ABB RAPID module: 001956CB

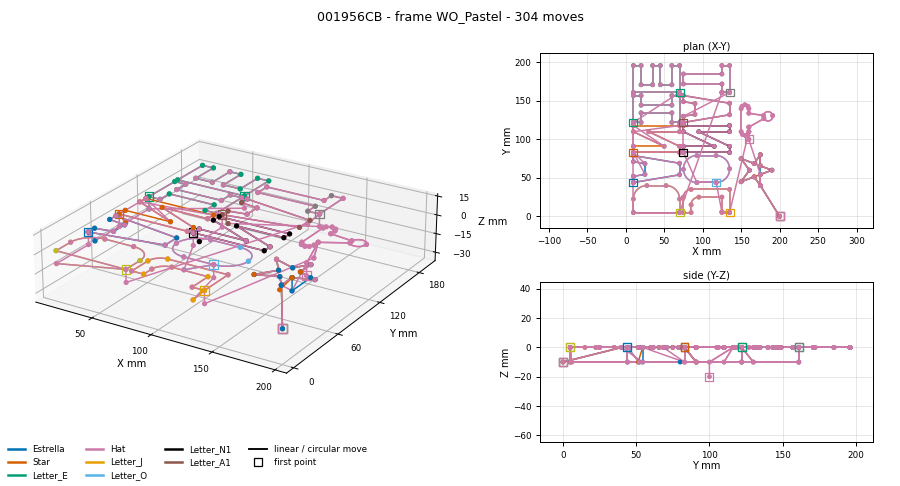
[picture p0: tool path of 001956CB in frame WO_Pastel, 304 of 314 moves have a stored position in this frame; points joined in program order, loops and branches not executed]
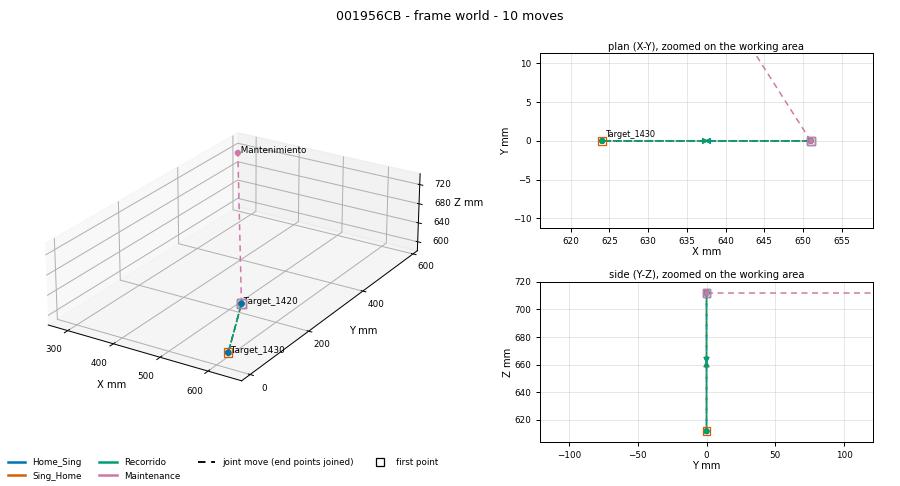
[picture p1: tool path of 001956CB in frame world, 10 of 314 moves have a stored position in this frame; points joined in program order, loops and branches not executed]
MODULE Module1
        CONST robtarget Target_10:=[[200,0,-10],[1,0,0,0],[0,0,2,0],[9E+09,9E+09,9E+09,9E+09,9E+09,9E+09]];
    CONST robtarget Target_20:=[[175,40,0],[1,0,0,0],[0,0,2,0],[9E+09,9E+09,9E+09,9E+09,9E+09,9E+09]];
    CONST robtarget Target_30:=[[175,54.375,0],[1,0,0,0],[0,0,2,0],[9E+09,9E+09,9E+09,9E+09,9E+09,9E+09]];
    CONST robtarget Target_40:=[[190,60,0],[1,0,0,0],[0,0,2,0],[9E+09,9E+09,9E+09,9E+09,9E+09,9E+09]];
    CONST robtarget Target_50:=[[175,65.625,0],[1,0,0,0],[0,0,2,0],[9E+09,9E+09,9E+09,9E+09,9E+09,9E+09]];
    CONST robtarget Target_60:=[[175,80,0],[1,0,0,0],[0,0,2,0],[9E+09,9E+09,9E+09,9E+09,9E+09,9E+09]];
    CONST robtarget Target_70:=[[166.901,68.662,0],[1,0,0,0],[0,0,2,0],[9E+09,9E+09,9E+09,9E+09,9E+09,9E+09]];
    CONST robtarget Target_80:=[[150,75,0],[1,0,0,0],[0,0,2,0],[9E+09,9E+09,9E+09,9E+09,9E+09,9E+09]];
    CONST robtarget Target_90:=[[160.714,60,0],[1,0,0,0],[0,0,2,0],[9E+09,9E+09,9E+09,9E+09,9E+09,9E+09]];
    CONST robtarget Target_100:=[[150,45,0],[1,0,0,0],[0,0,2,0],[9E+09,9E+09,9E+09,9E+09,9E+09,9E+09]];
    CONST robtarget Target_110:=[[166.901,51.338,0],[1,0,0,0],[0,0,2,0],[9E+09,9E+09,9E+09,9E+09,9E+09,9E+09]];
    CONST robtarget Target_120:=[[166.901,51.338,-10],[1,0,0,0],[-1,-1,2,0],[9E+09,9E+09,9E+09,9E+09,9E+09,9E+09]];
    CONST robtarget Target_130:=[[160,116,0],[1,0,0,0],[0,0,2,0],[9E+09,9E+09,9E+09,9E+09,9E+09,9E+09]];
    CONST robtarget Target_140:=[[179.71,127.038,0],[1,0,0,0],[0,0,2,0],[9E+09,9E+09,9E+09,9E+09,9E+09,9E+09]];
    CONST robtarget Target_150:=[[186.774,124.203,0],[1,0,0,0],[0,0,2,0],[9E+09,9E+09,9E+09,9E+09,9E+09,9E+09]];
    CONST robtarget Target_160:=[[190.983,130.98,0],[1,0,0,0],[0,0,2,0],[9E+09,9E+09,9E+09,9E+09,9E+09,9E+09]];
    CONST robtarget Target_170:=[[183.755,135.933,0],[1,0,0,0],[0,0,2,0],[9E+09,9E+09,9E+09,9E+09,9E+09,9E+09]];
    CONST robtarget Target_180:=[[179.014,130.957,0],[1,0,0,0],[0,0,2,0],[9E+09,9E+09,9E+09,9E+09,9E+09,9E+09]];
    CONST robtarget Target_190:=[[160,134,0],[1,0,0,0],[0,0,2,0],[9E+09,9E+09,9E+09,9E+09,9E+09,9E+09]];
    CONST robtarget Target_200:=[[160,140,0],[1,0,0,0],[0,0,2,0],[9E+09,9E+09,9E+09,9E+09,9E+09,9E+09]];
    CONST robtarget Target_210:=[[158.829,143.215,0],[1,0,0,0],[0,0,2,0],[9E+09,9E+09,9E+09,9E+09,9E+09,9E+09]];
    CONST robtarget Target_220:=[[154.832,144.997,0],[1,0,0,0],[0,0,2,0],[9E+09,9E+09,9E+09,9E+09,9E+09,9E+09]];
    CONST robtarget Target_230:=[[151.042,143.055,0],[1,0,0,0],[0,0,2,0],[9E+09,9E+09,9E+09,9E+09,9E+09,9E+09]];
        CONST robtarget HomeManipulador:=[[651,-0.02,712.04],[0.707129,-3.57758E-05,0.707084,6.57305E-06],[0,0,-1,0],[9E+09,9E+09,9E+09,9E+09,9E+09,9E+09]];
    CONST robtarget Target_1280:=[[70,161,0],[1,0,0,0],[-1,-2,-1,0],[9E+09,9E+09,9E+09,9E+09,9E+09,9E+09]];
    CONST robtarget Target_1290:=[[70,196,0],[1,0,0,0],[-1,-2,-1,0],[9E+09,9E+09,9E+09,9E+09,9E+09,9E+09]];
    CONST robtarget Target_1300:=[[60,196,0],[1,0,0,0],[-1,-2,-1,0],[9E+09,9E+09,9E+09,9E+09,9E+09,9E+09]];
    CONST robtarget Target_1310:=[[60,171,0],[1,0,0,0],[-1,-2,-1,0],[9E+09,9E+09,9E+09,9E+09,9E+09,9E+09]];
    CONST robtarget Target_1320:=[[45,171,0],[1,0,0,0],[-1,-2,-1,0],[9E+09,9E+09,9E+09,9E+09,9E+09,9E+09]];
    CONST robtarget Target_1330:=[[45,196,0],[1,0,0,0],[-1,-2,-1,0],[9E+09,9E+09,9E+09,9E+09,9E+09,9E+09]];
    CONST robtarget Target_1340:=[[35,196,0],[1,0,0,0],[-1,-2,-1,0],[9E+09,9E+09,9E+09,9E+09,9E+09,9E+09]];
    CONST robtarget Target_1350:=[[35,171,0],[1,0,0,0],[-1,-2,-1,0],[9E+09,9E+09,9E+09,9E+09,9E+09,9E+09]];
    CONST robtarget Target_1360:=[[20,171,0],[1,0,0,0],[-1,-2,-1,0],[9E+09,9E+09,9E+09,9E+09,9E+09,9E+09]];
    CONST robtarget Target_1370:=[[20,196,0],[1,0,0,0],[-1,-2,-1,0],[9E+09,9E+09,9E+09,9E+09,9E+09,9E+09]];
    CONST robtarget Target_1380:=[[10,196,0],[1,0,0,0],[-1,-2,-1,0],[9E+09,9E+09,9E+09,9E+09,9E+09,9E+09]];
    CONST robtarget Target_1390:=[[10,161,0],[1,0,0,0],[-1,-2,-1,0],[9E+09,9E+09,9E+09,9E+09,9E+09,9E+09]];
    CONST robtarget Target_1470:=[[160,100.007,-20],[1,0,0,0],[0,2,0,1],[9E+09,9E+09,9E+09,9E+09,9E+09,9E+09]];
    CONST robtarget Target_1440:=[[160,100,-10],[1,0,0,0],[0,0,2,0],[9E+09,9E+09,9E+09,9E+09,9E+09,9E+09]];
    CONST robtarget Target_240:=[[150,140,0],[1,0,0,0],[0,0,2,0],[9E+09,9E+09,9E+09,9E+09,9E+09,9E+09]];
    CONST robtarget Target_250:=[[150,110,0],[1,0,0,0],[0,0,2,0],[9E+09,9E+09,9E+09,9E+09,9E+09,9E+09]];
    CONST robtarget Target_260:=[[151.712,106.233,0],[1,0,0,0],[0,-1,2,0],[9E+09,9E+09,9E+09,9E+09,9E+09,9E+09]];
    CONST robtarget Target_270:=[[155.472,105.022,0],[1,0,0,0],[0,0,2,0],[9E+09,9E+09,9E+09,9E+09,9E+09,9E+09]];
    CONST robtarget Target_280:=[[158.325,106.266,0],[1,0,0,0],[0,0,2,0],[9E+09,9E+09,9E+09,9E+09,9E+09,9E+09]];
    CONST robtarget Target_290:=[[160,110.007,0],[1,0,0,0],[0,0,2,0],[9E+09,9E+09,9E+09,9E+09,9E+09,9E+09]];
    CONST robtarget Target_300:=[[160,110.007,-10],[1,0,0,0],[0,0,2,0],[9E+09,9E+09,9E+09,9E+09,9E+09,9E+09]];
    CONST robtarget Target_310_2:=[[135,5,0],[1,0,0,0],[0,0,2,0],[9E+09,9E+09,9E+09,9E+09,9E+09,9E+09]];
    CONST robtarget Target_320_2:=[[135,35,0],[1,0,0,0],[0,0,2,0],[9E+09,9E+09,9E+09,9E+09,9E+09,9E+09]];
    CONST robtarget Target_330_2:=[[85,35,0],[1,0,0,0],[0,0,2,0],[9E+09,9E+09,9E+09,9E+09,9E+09,9E+09]];
    CONST robtarget Target_340_2:=[[77.06,31.078,0],[1,0,0,0],[0,0,2,0],[9E+09,9E+09,9E+09,9E+09,9E+09,9E+09]];
    CONST robtarget Target_350_2:=[[75,25,0],[1,0,0,0],[0,0,2,0],[9E+09,9E+09,9E+09,9E+09,9E+09,9E+09]];
    CONST robtarget Target_360_2:=[[75,5,0],[1,0,0,0],[0,0,2,0],[9E+09,9E+09,9E+09,9E+09,9E+09,9E+09]];
    CONST robtarget Target_370_2:=[[85,5,0],[1,0,0,0],[0,0,2,0],[9E+09,9E+09,9E+09,9E+09,9E+09,9E+09]];
    CONST robtarget Target_380_2:=[[85,15,0],[1,0,0,0],[0,0,2,0],[9E+09,9E+09,9E+09,9E+09,9E+09,9E+09]];
    CONST robtarget Target_390_2:=[[87.41,21.51,0],[1,0,0,0],[0,0,2,0],[9E+09,9E+09,9E+09,9E+09,9E+09,9E+09]];
    CONST robtarget Target_400_2:=[[95,25,0],[1,0,0,0],[0,0,2,0],[9E+09,9E+09,9E+09,9E+09,9E+09,9E+09]];
    CONST robtarget Target_410_2:=[[125,25,0],[1,0,0,0],[0,0,2,0],[9E+09,9E+09,9E+09,9E+09,9E+09,9E+09]];
    CONST robtarget Target_420_2:=[[125,5,0],[1,0,0,0],[0,0,2,0],[9E+09,9E+09,9E+09,9E+09,9E+09,9E+09]];
    CONST robtarget Target_430_2:=[[125,6,-10],[1,0,0,0],[0,0,2,0],[9E+09,9E+09,9E+09,9E+09,9E+09,9E+09]];
    CONST robtarget Target_440:=[[117.496,44,0],[1,0,0,0],[0,0,2,0],[9E+09,9E+09,9E+09,9E+09,9E+09,9E+09]];
    CONST robtarget Target_450:=[[130.812,50.14,0],[1,0,0,0],[0,0,2,0],[9E+09,9E+09,9E+09,9E+09,9E+09,9E+09]];
    CONST robtarget Target_460:=[[134.997,61.803,0],[1,0,0,0],[0,0,2,0],[9E+09,9E+09,9E+09,9E+09,9E+09,9E+09]];
    CONST robtarget Target_470:=[[131.095,72.519,0],[1,0,0,0],[0,0,2,0],[9E+09,9E+09,9E+09,9E+09,9E+09,9E+09]];
    CONST robtarget Target_490:=[[117.5,79,0],[1,0,0,0],[0,0,2,0],[9E+09,9E+09,9E+09,9E+09,9E+09,9E+09]];
    CONST robtarget Target_500:=[[92.5,79,0],[1,0,0,0],[0,0,2,0],[9E+09,9E+09,9E+09,9E+09,9E+09,9E+09]];
    CONST robtarget Target_510:=[[80.951,74.647,0],[1,0,0,0],[0,0,2,0],[9E+09,9E+09,9E+09,9E+09,9E+09,9E+09]];
    CONST robtarget Target_520:=[[75.005,61.068,0],[1,0,0,0],[0,0,2,0],[9E+09,9E+09,9E+09,9E+09,9E+09,9E+09]];
    CONST robtarget Target_530:=[[79.917,49.337,0],[1,0,0,0],[0,0,2,0],[9E+09,9E+09,9E+09,9E+09,9E+09,9E+09]];
    CONST robtarget Target_550:=[[92.504,44,0],[1,0,0,0],[0,0,2,0],[9E+09,9E+09,9E+09,9E+09,9E+09,9E+09]];
    CONST robtarget Target_560:=[[92.504,44,-10],[1,0,0,0],[0,0,2,0],[9E+09,9E+09,9E+09,9E+09,9E+09,9E+09]];
    CONST robtarget Target_570:=[[75,83,0],[1,0,0,0],[0,0,2,0],[9E+09,9E+09,9E+09,9E+09,9E+09,9E+09]];
    CONST robtarget Target_580:=[[135,83,0],[1,0,0,0],[0,0,2,0],[9E+09,9E+09,9E+09,9E+09,9E+09,9E+09]];
    CONST robtarget Target_590:=[[135,91,0],[1,0,0,0],[0,0,2,0],[9E+09,9E+09,9E+09,9E+09,9E+09,9E+09]];
    CONST robtarget Target_600:=[[95,110,0],[1,0,0,0],[0,0,2,0],[9E+09,9E+09,9E+09,9E+09,9E+09,9E+09]];
    CONST robtarget Target_610:=[[135,110,0],[1,0,0,0],[0,0,2,0],[9E+09,9E+09,9E+09,9E+09,9E+09,9E+09]];
    CONST robtarget Target_620:=[[135,118,0],[1,0,0,0],[0,0,2,0],[9E+09,9E+09,9E+09,9E+09,9E+09,9E+09]];
    CONST robtarget Target_630:=[[75,118,0],[1,0,0,0],[0,0,2,0],[9E+09,9E+09,9E+09,9E+09,9E+09,9E+09]];
    CONST robtarget Target_640:=[[75,110,0],[1,0,0,0],[0,0,2,0],[9E+09,9E+09,9E+09,9E+09,9E+09,9E+09]];
    CONST robtarget Target_650:=[[115,91,0],[1,0,0,0],[0,0,2,0],[9E+09,9E+09,9E+09,9E+09,9E+09,9E+09]];
    CONST robtarget Target_660:=[[75,91,0],[1,0,0,0],[0,0,2,0],[9E+09,9E+09,9E+09,9E+09,9E+09,9E+09]];
    CONST robtarget Target_670:=[[75,91,-10],[1,0,0,0],[0,0,2,0],[9E+09,9E+09,9E+09,9E+09,9E+09,9E+09]];
    CONST robtarget Target_680:=[[75,122,0],[1,0,0,0],[0,0,2,0],[9E+09,9E+09,9E+09,9E+09,9E+09,9E+09]];
    CONST robtarget Target_690:=[[135,132,0],[1,0,0,0],[0,0,2,0],[9E+09,9E+09,9E+09,9E+09,9E+09,9E+09]];
    CONST robtarget Target_700:=[[135,147,0],[1,0,0,0],[0,0,2,0],[9E+09,9E+09,9E+09,9E+09,9E+09,9E+09]];
    CONST robtarget Target_710:=[[75,157,0],[1,0,0,0],[0,0,2,0],[9E+09,9E+09,9E+09,9E+09,9E+09,9E+09]];
    CONST robtarget Target_720:=[[75,149,0],[1,0,0,0],[0,0,2,0],[9E+09,9E+09,9E+09,9E+09,9E+09,9E+09]];
    CONST robtarget Target_730:=[[90,146.5,0],[1,0,0,0],[0,0,2,0],[9E+09,9E+09,9E+09,9E+09,9E+09,9E+09]];
    CONST robtarget Target_740:=[[90,132.5,0],[1,0,0,0],[0,0,2,0],[9E+09,9E+09,9E+09,9E+09,9E+09,9E+09]];
    CONST robtarget Target_750:=[[75,130,0],[1,0,0,0],[0,0,2,0],[9E+09,9E+09,9E+09,9E+09,9E+09,9E+09]];
    CONST robtarget Target_760:=[[75,130,-10],[1,0,0,0],[0,0,2,0],[9E+09,9E+09,9E+09,9E+09,9E+09,9E+09]];
    CONST robtarget Target_770:=[[135,161,0],[1,0,0,0],[0,0,2,0],[9E+09,9E+09,9E+09,9E+09,9E+09,9E+09]];
    CONST robtarget Target_780:=[[135,196,0],[1,0,0,0],[0,0,2,0],[9E+09,9E+09,9E+09,9E+09,9E+09,9E+09]];
    CONST robtarget Target_790:=[[125,196,0],[1,0,0,0],[0,0,2,0],[9E+09,9E+09,9E+09,9E+09,9E+09,9E+09]];
    CONST robtarget Target_800:=[[125,185,0],[1,0,0,0],[0,0,2,0],[9E+09,9E+09,9E+09,9E+09,9E+09,9E+09]];
    CONST robtarget Target_810:=[[75,185,0],[1,0,0,0],[0,0,2,0],[9E+09,9E+09,9E+09,9E+09,9E+09,9E+09]];
    CONST robtarget Target_820:=[[75,172,0],[1,0,0,0],[0,0,2,0],[9E+09,9E+09,9E+09,9E+09,9E+09,9E+09]];
    CONST robtarget Target_830:=[[125,172,0],[1,0,0,0],[0,0,2,0],[9E+09,9E+09,9E+09,9E+09,9E+09,9E+09]];
    CONST robtarget Target_840:=[[125,161,0],[1,0,0,0],[0,0,2,0],[9E+09,9E+09,9E+09,9E+09,9E+09,9E+09]];
    CONST robtarget Target_850:=[[125,161,-10],[1,0,0,0],[0,0,2,0],[9E+09,9E+09,9E+09,9E+09,9E+09,9E+09]];
    CONST robtarget Target_860:=[[70,5,0],[1,0,0,0],[0,0,2,0],[9E+09,9E+09,9E+09,9E+09,9E+09,9E+09]];
    CONST robtarget Target_870:=[[70,22.489,0],[1,0,0,0],[0,0,2,0],[9E+09,9E+09,9E+09,9E+09,9E+09,9E+09]];
    CONST robtarget Target_880:=[[65.387,34.34,0],[1,0,0,0],[0,0,2,0],[9E+09,9E+09,9E+09,9E+09,9E+09,9E+09]];
    CONST robtarget Target_890:=[[52.5,40,0],[1,0,0,0],[0,0,2,0],[9E+09,9E+09,9E+09,9E+09,9E+09,9E+09]];
    CONST robtarget Target_900:=[[27.5,40,0],[1,0,0,0],[0,0,2,0],[9E+09,9E+09,9E+09,9E+09,9E+09,9E+09]];
    CONST robtarget Target_910:=[[14.273,33.958,0],[1,0,0,0],[0,0,2,0],[9E+09,9E+09,9E+09,9E+09,9E+09,9E+09]];
    CONST robtarget Target_920:=[[10,22.489,0],[1,0,0,0],[0,-1,2,0],[9E+09,9E+09,9E+09,9E+09,9E+09,9E+09]];
    CONST robtarget Target_930:=[[10,5,0],[1,0,0,0],[0,0,2,0],[9E+09,9E+09,9E+09,9E+09,9E+09,9E+09]];
    CONST robtarget Target_940:=[[10,5,-10],[1,0,0,0],[0,0,2,0],[9E+09,9E+09,9E+09,9E+09,9E+09,9E+09]];
    CONST robtarget Target_950:=[[10,44,0],[1,0,0,0],[0,0,2,0],[9E+09,9E+09,9E+09,9E+09,9E+09,9E+09]];
    CONST robtarget Target_960:=[[70,54,0],[1,0,0,0],[0,0,2,0],[9E+09,9E+09,9E+09,9E+09,9E+09,9E+09]];
    CONST robtarget Target_970:=[[70,69,0],[1,0,0,0],[0,0,2,0],[9E+09,9E+09,9E+09,9E+09,9E+09,9E+09]];
    CONST robtarget Target_980:=[[10,79,0],[1,0,0,0],[0,0,2,0],[9E+09,9E+09,9E+09,9E+09,9E+09,9E+09]];
    CONST robtarget Target_990:=[[10,71,0],[1,0,0,0],[0,0,2,0],[9E+09,9E+09,9E+09,9E+09,9E+09,9E+09]];
    CONST robtarget Target_1000:=[[25,68.5,0],[1,0,0,0],[0,0,2,0],[9E+09,9E+09,9E+09,9E+09,9E+09,9E+09]];
    CONST robtarget Target_1010:=[[25,54.5,0],[1,0,0,0],[0,0,2,0],[9E+09,9E+09,9E+09,9E+09,9E+09,9E+09]];
    CONST robtarget Target_1020:=[[10,52,0],[1,0,0,0],[0,0,2,0],[9E+09,9E+09,9E+09,9E+09,9E+09,9E+09]];
    CONST robtarget Target_1030:=[[10,52,-10],[1,0,0,0],[0,0,2,0],[9E+09,9E+09,9E+09,9E+09,9E+09,9E+09]];
    CONST robtarget Target_1040:=[[10,83,0],[1,0,0,0],[0,0,2,0],[9E+09,9E+09,9E+09,9E+09,9E+09,9E+09]];
    CONST robtarget Target_1050:=[[70,83,0],[1,0,0,0],[0,0,2,0],[9E+09,9E+09,9E+09,9E+09,9E+09,9E+09]];
    CONST robtarget Target_1060:=[[70,91,0],[1,0,0,0],[0,0,2,0],[9E+09,9E+09,9E+09,9E+09,9E+09,9E+09]];
    CONST robtarget Target_1070:=[[30,110,0],[1,0,0,0],[0,0,2,0],[9E+09,9E+09,9E+09,9E+09,9E+09,9E+09]];
    CONST robtarget Target_1080:=[[70,110,0],[1,0,0,0],[0,0,2,0],[9E+09,9E+09,9E+09,9E+09,9E+09,9E+09]];
    CONST robtarget Target_1090:=[[70,118,0],[1,0,0,0],[0,0,2,0],[9E+09,9E+09,9E+09,9E+09,9E+09,9E+09]];
    CONST robtarget Target_1100:=[[10,118,0],[1,0,0,0],[0,0,2,0],[9E+09,9E+09,9E+09,9E+09,9E+09,9E+09]];
    CONST robtarget Target_1110:=[[10,110,0],[1,0,0,0],[0,0,2,0],[9E+09,9E+09,9E+09,9E+09,9E+09,9E+09]];
    CONST robtarget Target_1120:=[[50,91,0],[1,0,0,0],[0,0,2,0],[9E+09,9E+09,9E+09,9E+09,9E+09,9E+09]];
    CONST robtarget Target_1130:=[[10,91,0],[1,0,0,0],[0,0,2,0],[9E+09,9E+09,9E+09,9E+09,9E+09,9E+09]];
    CONST robtarget Target_1140:=[[10,91,-10],[1,0,0,0],[0,0,2,0],[9E+09,9E+09,9E+09,9E+09,9E+09,9E+09]];
    CONST robtarget Target_1150:=[[10,122,0],[1,0,0,0],[-1,-2,-1,0],[9E+09,9E+09,9E+09,9E+09,9E+09,9E+09]];
    CONST robtarget Target_1160:=[[20,122,0],[1,0,0,0],[-1,-2,-1,0],[9E+09,9E+09,9E+09,9E+09,9E+09,9E+09]];
    CONST robtarget Target_1170:=[[20,134.5,0],[1,0,0,0],[-1,-2,-1,0],[9E+09,9E+09,9E+09,9E+09,9E+09,9E+09]];
    CONST robtarget Target_1180:=[[60,134.5,0],[1,0,0,0],[-1,-2,-1,0],[9E+09,9E+09,9E+09,9E+09,9E+09,9E+09]];
    CONST robtarget Target_1190:=[[60,122,0],[1,0,0,0],[-1,-2,-1,0],[9E+09,9E+09,9E+09,9E+09,9E+09,9E+09]];
    CONST robtarget Target_1200:=[[70,122,0],[1,0,0,0],[-1,-1,-1,0],[9E+09,9E+09,9E+09,9E+09,9E+09,9E+09]];
    CONST robtarget Target_1210:=[[70,157,0],[1,0,0,0],[-1,-2,-1,0],[9E+09,9E+09,9E+09,9E+09,9E+09,9E+09]];
    CONST robtarget Target_1220:=[[60,157,0],[1,0,0,0],[-1,-2,-1,0],[9E+09,9E+09,9E+09,9E+09,9E+09,9E+09]];
    CONST robtarget Target_1230:=[[60,144.5,0],[1,0,0,0],[-1,-2,-1,0],[9E+09,9E+09,9E+09,9E+09,9E+09,9E+09]];
    CONST robtarget Target_1240:=[[20,144.5,0],[1,0,0,0],[-1,-2,-1,0],[9E+09,9E+09,9E+09,9E+09,9E+09,9E+09]];
    CONST robtarget Target_1250:=[[20,157,0],[1,0,0,0],[-1,-2,-1,0],[9E+09,9E+09,9E+09,9E+09,9E+09,9E+09]];
    CONST robtarget Target_1260:=[[10,157,0],[1,0,0,0],[-1,-2,-1,0],[9E+09,9E+09,9E+09,9E+09,9E+09,9E+09]];
    CONST robtarget Target_1270:=[[10,122,-10],[1,0,0,0],[0,0,2,0],[9E+09,9E+09,9E+09,9E+09,9E+09,9E+09]];
    CONST robtarget Target_1420:=[[651.002006649,-0.016010457,712.036997271],[0.707129293,-0.000035776,0.707084268,0.000006573],[0,-1,-1,0],[9E+09,9E+09,9E+09,9E+09,9E+09,9E+09]];
    CONST robtarget Target_1430:=[[624.074169941,-0.017623285,611.525498045],[0.500005745,-0.00004382,0.866022086,0.000004646],[0,-1,-1,0],[9E+09,9E+09,9E+09,9E+09,9E+09,9E+09]];
    CONST robtarget Target_1460:=[[175,80,-10],[1,0,0,0],[0,0,2,0],[9E+09,9E+09,9E+09,9E+09,9E+09,9E+09]];
    CONST robtarget Target_1450:=[[175,54.375,-10],[1,0,0,0],[0,0,2,0],[9E+09,9E+09,9E+09,9E+09,9E+09,9E+09]];
    CONST robtarget Target_1480:=[[135,5,-10],[1,0,0,0],[0,0,2,0],[9E+09,9E+09,9E+09,9E+09,9E+09,9E+09]];
    CONST robtarget Target_310:=[[135,5,0],[1,0,0,0],[0,0,2,0],[9E+09,9E+09,9E+09,9E+09,9E+09,9E+09]];
    CONST robtarget Target_320:=[[135,35,0],[1,0,0,0],[0,0,2,0],[9E+09,9E+09,9E+09,9E+09,9E+09,9E+09]];
    CONST robtarget Target_330:=[[85,35,0],[1,0,0,0],[0,0,2,0],[9E+09,9E+09,9E+09,9E+09,9E+09,9E+09]];
    CONST robtarget Target_340:=[[77.06,31.078,0],[1,0,0,0],[0,0,2,0],[9E+09,9E+09,9E+09,9E+09,9E+09,9E+09]];
    CONST robtarget Target_350:=[[75,25,0],[1,0,0,0],[0,0,2,0],[9E+09,9E+09,9E+09,9E+09,9E+09,9E+09]];
    CONST robtarget Target_360:=[[75,5,0],[1,0,0,0],[0,0,2,0],[9E+09,9E+09,9E+09,9E+09,9E+09,9E+09]];
    CONST robtarget Target_370:=[[85,5,0],[1,0,0,0],[0,0,2,0],[9E+09,9E+09,9E+09,9E+09,9E+09,9E+09]];
    CONST robtarget Target_380:=[[85,15,0],[1,0,0,0],[0,0,2,0],[9E+09,9E+09,9E+09,9E+09,9E+09,9E+09]];
    CONST robtarget Target_390:=[[87.41,21.51,0],[1,0,0,0],[0,0,2,0],[9E+09,9E+09,9E+09,9E+09,9E+09,9E+09]];
    CONST robtarget Target_400:=[[95,25,0],[1,0,0,0],[0,0,2,0],[9E+09,9E+09,9E+09,9E+09,9E+09,9E+09]];
    CONST robtarget Target_410:=[[125,25,0],[1,0,0,0],[0,0,2,0],[9E+09,9E+09,9E+09,9E+09,9E+09,9E+09]];
    CONST robtarget Target_420:=[[125,5,0],[1,0,0,0],[0,0,2,0],[9E+09,9E+09,9E+09,9E+09,9E+09,9E+09]];
    CONST robtarget Target_430:=[[125,6,-10],[1,0,0,0],[0,0,2,0],[9E+09,9E+09,9E+09,9E+09,9E+09,9E+09]];
    CONST robtarget Target_1490:=[[117.496,44,-10],[1,0,0,0],[0,0,2,0],[9E+09,9E+09,9E+09,9E+09,9E+09,9E+09]];
    CONST robtarget Target_1500:=[[75,83,-10],[1,0,0,0],[0,0,2,0],[9E+09,9E+09,9E+09,9E+09,9E+09,9E+09]];
    CONST robtarget Target_1510:=[[75,122,-10],[1,0,0,0],[0,0,2,0],[9E+09,9E+09,9E+09,9E+09,9E+09,9E+09]];
    CONST robtarget Target_1520:=[[135,161,-10],[1,0,0,0],[0,0,2,0],[9E+09,9E+09,9E+09,9E+09,9E+09,9E+09]];
    CONST robtarget Target_1530:=[[70,5,-10],[1,0,0,0],[0,0,2,0],[9E+09,9E+09,9E+09,9E+09,9E+09,9E+09]];
    CONST robtarget Target_1540:=[[10,44,-10],[1,0,0,0],[0,0,2,0],[9E+09,9E+09,9E+09,9E+09,9E+09,9E+09]];
    CONST robtarget Target_1550:=[[10,83,-10],[1,0,0,0],[0,0,2,0],[9E+09,9E+09,9E+09,9E+09,9E+09,9E+09]];
    CONST robtarget Target_1150_2:=[[10,122,0],[1,0,0,0],[0,0,2,0],[9E+09,9E+09,9E+09,9E+09,9E+09,9E+09]];
    CONST robtarget Target_1160_2:=[[20,122,0],[1,0,0,0],[0,0,2,0],[9E+09,9E+09,9E+09,9E+09,9E+09,9E+09]];
    CONST robtarget Target_1170_2:=[[20,134.5,0],[1,0,0,0],[0,0,2,0],[9E+09,9E+09,9E+09,9E+09,9E+09,9E+09]];
    CONST robtarget Target_1180_2:=[[60,134.5,0],[1,0,0,0],[0,0,2,0],[9E+09,9E+09,9E+09,9E+09,9E+09,9E+09]];
    CONST robtarget Target_1190_2:=[[60,122,0],[1,0,0,0],[0,0,2,0],[9E+09,9E+09,9E+09,9E+09,9E+09,9E+09]];
    CONST robtarget Target_1200_2:=[[70,122,0],[1,0,0,0],[0,0,2,0],[9E+09,9E+09,9E+09,9E+09,9E+09,9E+09]];
    CONST robtarget Target_1210_2:=[[70,157,0],[1,0,0,0],[0,0,2,0],[9E+09,9E+09,9E+09,9E+09,9E+09,9E+09]];
    CONST robtarget Target_1220_2:=[[60,157,0],[1,0,0,0],[0,0,2,0],[9E+09,9E+09,9E+09,9E+09,9E+09,9E+09]];
    CONST robtarget Target_1230_2:=[[60,144.5,0],[1,0,0,0],[0,0,2,0],[9E+09,9E+09,9E+09,9E+09,9E+09,9E+09]];
    CONST robtarget Target_1240_2:=[[20,144.5,0],[1,0,0,0],[0,0,2,0],[9E+09,9E+09,9E+09,9E+09,9E+09,9E+09]];
    CONST robtarget Target_1250_2:=[[20,157,0],[1,0,0,0],[0,0,2,0],[9E+09,9E+09,9E+09,9E+09,9E+09,9E+09]];
    CONST robtarget Target_1260_2:=[[10,157,0],[1,0,0,0],[0,0,2,0],[9E+09,9E+09,9E+09,9E+09,9E+09,9E+09]];
    CONST robtarget Target_1270_2:=[[10,122,-10],[1,0,0,0],[0,0,2,0],[9E+09,9E+09,9E+09,9E+09,9E+09,9E+09]];
    CONST robtarget Target_1560:=[[70,161,-10],[1,0,0,0],[0,0,2,0],[9E+09,9E+09,9E+09,9E+09,9E+09,9E+09]];
    CONST robtarget Target_1280_2:=[[70,161,0],[1,0,0,0],[0,0,2,0],[9E+09,9E+09,9E+09,9E+09,9E+09,9E+09]];
    CONST robtarget Target_1290_2:=[[70,196,0],[1,0,0,0],[0,0,2,0],[9E+09,9E+09,9E+09,9E+09,9E+09,9E+09]];
    CONST robtarget Target_1300_2:=[[60,196,0],[1,0,0,0],[0,0,2,0],[9E+09,9E+09,9E+09,9E+09,9E+09,9E+09]];
    CONST robtarget Target_1310_2:=[[60,171,0],[1,0,0,0],[0,0,2,0],[9E+09,9E+09,9E+09,9E+09,9E+09,9E+09]];
    CONST robtarget Target_1320_2:=[[45,171,0],[1,0,0,0],[0,0,2,0],[9E+09,9E+09,9E+09,9E+09,9E+09,9E+09]];
    CONST robtarget Target_1330_2:=[[45,196,0],[1,0,0,0],[0,0,2,0],[9E+09,9E+09,9E+09,9E+09,9E+09,9E+09]];
    CONST robtarget Target_1340_2:=[[35,196,0],[1,0,0,0],[0,0,2,0],[9E+09,9E+09,9E+09,9E+09,9E+09,9E+09]];
    CONST robtarget Target_1350_2:=[[35,171,0],[1,0,0,0],[0,0,2,0],[9E+09,9E+09,9E+09,9E+09,9E+09,9E+09]];
    CONST robtarget Target_1360_2:=[[20,171,0],[1,0,0,0],[0,0,2,0],[9E+09,9E+09,9E+09,9E+09,9E+09,9E+09]];
    CONST robtarget Target_1370_2:=[[20,196,0],[1,0,0,0],[0,0,2,0],[9E+09,9E+09,9E+09,9E+09,9E+09,9E+09]];
    CONST robtarget Target_1380_2:=[[10,196,0],[1,0,0,0],[0,0,2,0],[9E+09,9E+09,9E+09,9E+09,9E+09,9E+09]];
    CONST robtarget Target_1390_2:=[[10,161,0],[1,0,0,0],[0,0,2,0],[9E+09,9E+09,9E+09,9E+09,9E+09,9E+09]];
    CONST robtarget Mantenimiento:=[[274.21719642,590.430860773,712.037008126],[0.596086109,-0.380412267,0.596032433,0.380411878],[0,0,-1,0],[9E+09,9E+09,9E+09,9E+09,9E+09,9E+09]];
!***********************************************************
    !
    ! M?dulo:  Module1
    !
    ! Descripci?n:
    !   <Introduzca la descripci?n aqu?>
    !
    ! Autor: jonaj
    !
    ! Versi?n: 1.0
    !
    !***********************************************************


    !***********************************************************
    !
    ! Procedimiento Main
    !
    !   Este es el punto de entrada de su programa
    !
    !*********************************************************** abb robotstudio tool definition with tcp & z
    PROC main()
        !Add your code here
        WHILE TRUE DO
            IF DI_01=1 THEN
                SetDO DO_01,1;
                Recorrido;
                SetDO DO_01,0;
            ELSEIF DI_02=1 THEN
                SetDO DO_02,1;
                Maintenance;
                SetDO DO_02,0;
            ENDIF
        ENDWHILE


        SetDO DO_02,1;
        Maintenance;
        SetDO DO_02,0;
    ENDPROC
    PROC Path_10()

    ENDPROC
    PROC Path_20()
    ENDPROC
    PROC Path_30()

    ENDPROC
    PROC Path_40()

    ENDPROC
    PROC Estrella()
        MoveL Target_10,v1000,z100,PortaMarcador\WObj:=WO_Pastel;
        MoveL Target_20,v1000,fine,PortaMarcador\WObj:=WO_Pastel;
        MoveL Target_30,v1000,fine,PortaMarcador\WObj:=WO_Pastel;
        MoveL Target_40,v1000,fine,PortaMarcador\WObj:=WO_Pastel;
        MoveL Target_50,v1000,fine,PortaMarcador\WObj:=WO_Pastel;
        MoveL Target_60,v1000,fine,PortaMarcador\WObj:=WO_Pastel;
        MoveL Target_70,v1000,fine,PortaMarcador\WObj:=WO_Pastel;
        MoveL Target_80,v1000,fine,PortaMarcador\WObj:=WO_Pastel;
        MoveL Target_90,v1000,fine,PortaMarcador\WObj:=WO_Pastel;
        MoveL Target_100,v1000,fine,PortaMarcador\WObj:=WO_Pastel;
        MoveL Target_110,v1000,fine,PortaMarcador\WObj:=WO_Pastel;
        MoveL Target_20,v1000,fine,PortaMarcador\WObj:=WO_Pastel;
        MoveL Target_30,v1000,fine,PortaMarcador\WObj:=WO_Pastel;
        MoveL Target_1450,v1000,z20,PortaMarcador\WObj:=WO_Pastel;
        MoveL Target_1460,v1000,z100,PortaMarcador\WObj:=WO_Pastel;
    ENDPROC
    PROC Star()
        MoveJ Target_10,v500,z100,PortaMarcador\WObj:=WO_Pastel;
        MoveL Target_20,v500,fine,PortaMarcador\WObj:=WO_Pastel;
        MoveL Target_30,v500,fine,PortaMarcador\WObj:=WO_Pastel;
        MoveL Target_40,v500,fine,PortaMarcador\WObj:=WO_Pastel;
        MoveL Target_50,v500,fine,PortaMarcador\WObj:=WO_Pastel;
        MoveL Target_60,v500,fine,PortaMarcador\WObj:=WO_Pastel;
        MoveL Target_70,v500,fine,PortaMarcador\WObj:=WO_Pastel;
        MoveL Target_80,v500,fine,PortaMarcador\WObj:=WO_Pastel;
        MoveL Target_90,v500,fine,PortaMarcador\WObj:=WO_Pastel;
        MoveL Target_100,v500,fine,PortaMarcador\WObj:=WO_Pastel;
        MoveL Target_110,v500,fine,PortaMarcador\WObj:=WO_Pastel;
        MoveL Target_20,v500,fine,PortaMarcador\WObj:=WO_Pastel;
        MoveL Target_30,v500,fine,PortaMarcador\WObj:=WO_Pastel;
        MoveL Target_120,v500,z100,PortaMarcador\WObj:=WO_Pastel;
    ENDPROC
    PROC Letter_E()
        MoveL Target_1280,v1000,z100,PortaMarcador\WObj:=WO_Pastel;
        MoveL Target_1290,v1000,fine,PortaMarcador\WObj:=WO_Pastel;
        MoveL Target_1300,v1000,fine,PortaMarcador\WObj:=WO_Pastel;
        MoveL Target_1310,v1000,fine,PortaMarcador\WObj:=WO_Pastel;
        MoveL Target_1320,v1000,fine,PortaMarcador\WObj:=WO_Pastel;
        MoveL Target_1330,v1000,fine,PortaMarcador\WObj:=WO_Pastel;
        MoveL Target_1340,v1000,fine,PortaMarcador\WObj:=WO_Pastel;
        MoveL Target_1350,v1000,fine,PortaMarcador\WObj:=WO_Pastel;
        MoveL Target_1360,v1000,fine,PortaMarcador\WObj:=WO_Pastel;
        MoveL Target_1370,v1000,fine,PortaMarcador\WObj:=WO_Pastel;
        MoveL Target_1380,v1000,fine,PortaMarcador\WObj:=WO_Pastel;
        MoveL Target_1390,v1000,z100,PortaMarcador\WObj:=WO_Pastel;
        MoveL Target_1280,v1000,z100,PortaMarcador\WObj:=WO_Pastel;
    ENDPROC
    PROC Hat()
        MoveL Target_1470,v1000,z40,PortaMarcador\WObj:=WO_Pastel;
        MoveL Target_1440,v1000,z15,PortaMarcador\WObj:=WO_Pastel;
        MoveL Target_130,v400,fine,PortaMarcador\WObj:=WO_Pastel;
        MoveL Target_140,v400,z10,PortaMarcador\WObj:=WO_Pastel;
        MoveC Target_150,Target_160,v400,z100,PortaMarcador\WObj:=WO_Pastel;
        MoveC Target_170,Target_180,v400,z100,PortaMarcador\WObj:=WO_Pastel;
        MoveL Target_190,v400,fine,PortaMarcador\WObj:=WO_Pastel;
        MoveL Target_200,v400,z100,PortaMarcador\WObj:=WO_Pastel;
        MoveL Target_210,v400,z100,PortaMarcador\WObj:=WO_Pastel;
        MoveL Target_220,v400,z100,PortaMarcador\WObj:=WO_Pastel;
        MoveL Target_230,v400,z100,PortaMarcador\WObj:=WO_Pastel;
        MoveL Target_240,v400,z100,PortaMarcador\WObj:=WO_Pastel;
        MoveL Target_250,v400,z100,PortaMarcador\WObj:=WO_Pastel;
        MoveL Target_260,v400,z100,PortaMarcador\WObj:=WO_Pastel;
        MoveL Target_270,v400,z100,PortaMarcador\WObj:=WO_Pastel;
        MoveL Target_280,v400,z100,PortaMarcador\WObj:=WO_Pastel;
        MoveL Target_290,v400,z100,PortaMarcador\WObj:=WO_Pastel;
        MoveL Target_130,v400,fine,PortaMarcador\WObj:=WO_Pastel;
        MoveL Target_300,v400,z100,PortaMarcador\WObj:=WO_Pastel;
    ENDPROC
    PROC Letter_J()
        MoveL Target_310_2,v50,z100,PortaMarcador\WObj:=WO_Pastel;
        MoveL Target_320_2,v50,fine,PortaMarcador\WObj:=WO_Pastel;
        MoveL Target_330_2,v50,z100,PortaMarcador\WObj:=WO_Pastel;
        MoveC Target_340_2,Target_350_2,v50,z100,PortaMarcador\WObj:=WO_Pastel;
        MoveL Target_360_2,v50,fine,PortaMarcador\WObj:=WO_Pastel;
        MoveL Target_370_2,v50,fine,PortaMarcador\WObj:=WO_Pastel;
        MoveL Target_380_2,v50,z100,PortaMarcador\WObj:=WO_Pastel;
        MoveC Target_390_2,Target_400_2,v50,z100,PortaMarcador\WObj:=WO_Pastel;
        MoveL Target_410_2,v50,fine,PortaMarcador\WObj:=WO_Pastel;
        MoveL Target_420_2,v50,fine,PortaMarcador\WObj:=WO_Pastel;
        MoveL Target_310_2,v50,fine,PortaMarcador\WObj:=WO_Pastel;
        MoveL Target_430_2,v1000,z100,PortaMarcador\WObj:=WO_Pastel;
    ENDPROC
    PROC Letter_O()
        MoveL Target_440,v100,z100,PortaMarcador\WObj:=WO_Pastel;
        MoveC Target_450,Target_460,v100,z100,PortaMarcador\WObj:=WO_Pastel;
        MoveC Target_470,Target_490,v100,z100,PortaMarcador\WObj:=WO_Pastel;
        MoveL Target_500,v100,z100,PortaMarcador\WObj:=WO_Pastel;
        MoveC Target_510,Target_520,v100,z100,PortaMarcador\WObj:=WO_Pastel;
        MoveC Target_530,Target_550,v100,z100,PortaMarcador\WObj:=WO_Pastel;
        MoveL Target_440,v100,fine,PortaMarcador\WObj:=WO_Pastel;
        MoveL Target_560,v100,z100,PortaMarcador\WObj:=WO_Pastel;
    ENDPROC
    PROC Letter_N1()
        MoveL Target_570,v400,fine,PortaMarcador\WObj:=WO_Pastel;
        MoveL Target_580,v400,fine,PortaMarcador\WObj:=WO_Pastel;
        MoveL Target_590,v400,fine,PortaMarcador\WObj:=WO_Pastel;
        MoveL Target_600,v400,fine,PortaMarcador\WObj:=WO_Pastel;
        MoveL Target_610,v400,fine,PortaMarcador\WObj:=WO_Pastel;
        MoveL Target_620,v400,fine,PortaMarcador\WObj:=WO_Pastel;
        MoveL Target_630,v400,fine,PortaMarcador\WObj:=WO_Pastel;
        MoveL Target_640,v400,fine,PortaMarcador\WObj:=WO_Pastel;
        MoveL Target_650,v400,fine,PortaMarcador\WObj:=WO_Pastel;
        MoveL Target_660,v400,fine,PortaMarcador\WObj:=WO_Pastel;
        MoveL Target_570,v400,fine,PortaMarcador\WObj:=WO_Pastel;
        MoveL Target_670,v400,z100,PortaMarcador\WObj:=WO_Pastel;
    ENDPROC
    PROC Letter_A1()
        MoveL Target_680,v600,fine,PortaMarcador\WObj:=WO_Pastel;
        MoveL Target_690,v600,fine,PortaMarcador\WObj:=WO_Pastel;
        MoveL Target_700,v600,fine,PortaMarcador\WObj:=WO_Pastel;
        MoveL Target_710,v600,fine,PortaMarcador\WObj:=WO_Pastel;
        MoveL Target_720,v600,fine,PortaMarcador\WObj:=WO_Pastel;
        MoveL Target_730,v600,fine,PortaMarcador\WObj:=WO_Pastel;
        MoveL Target_740,v600,fine,PortaMarcador\WObj:=WO_Pastel;
        MoveL Target_750,v600,fine,PortaMarcador\WObj:=WO_Pastel;
        MoveL Target_680,v600,fine,PortaMarcador\WObj:=WO_Pastel;
        MoveL Target_760,v600,fine,PortaMarcador\WObj:=WO_Pastel;
    ENDPROC
    PROC Letter_T()
        MoveL Target_770,v1000,fine,PortaMarcador\WObj:=WO_Pastel;
        MoveL Target_780,v1000,fine,PortaMarcador\WObj:=WO_Pastel;
        MoveL Target_790,v1000,fine,PortaMarcador\WObj:=WO_Pastel;
        MoveL Target_800,v1000,fine,PortaMarcador\WObj:=WO_Pastel;
        MoveL Target_810,v1000,fine,PortaMarcador\WObj:=WO_Pastel;
        MoveL Target_820,v1000,fine,PortaMarcador\WObj:=WO_Pastel;
        MoveL Target_830,v1000,fine,PortaMarcador\WObj:=WO_Pastel;
        MoveL Target_840,v1000,fine,PortaMarcador\WObj:=WO_Pastel;
        MoveL Target_770,v1000,fine,PortaMarcador\WObj:=WO_Pastel;
        MoveL Target_850,v1000,z100,PortaMarcador\WObj:=WO_Pastel;
    ENDPROC
    PROC Letter_D()
        MoveL Target_860,v1000,fine,PortaMarcador\WObj:=WO_Pastel;
        MoveL Target_870,v1000,fine,PortaMarcador\WObj:=WO_Pastel;
        MoveC Target_880,Target_890,v1000,fine,PortaMarcador\WObj:=WO_Pastel;
        MoveL Target_900,v1000,fine,PortaMarcador\WObj:=WO_Pastel;
        MoveC Target_910,Target_920,v1000,fine,PortaMarcador\WObj:=WO_Pastel;
        MoveL Target_930,v1000,fine,PortaMarcador\WObj:=WO_Pastel;
        MoveL Target_860,v1000,fine,PortaMarcador\WObj:=WO_Pastel;
        MoveL Target_940,v1000,z100,PortaMarcador\WObj:=WO_Pastel;
    ENDPROC
    PROC Letter_A2()
        MoveL Target_950,v1000,fine,PortaMarcador\WObj:=WO_Pastel;
        MoveL Target_960,v1000,fine,PortaMarcador\WObj:=WO_Pastel;
        MoveL Target_970,v1000,fine,PortaMarcador\WObj:=WO_Pastel;
        MoveL Target_980,v1000,fine,PortaMarcador\WObj:=WO_Pastel;
        MoveL Target_990,v1000,fine,PortaMarcador\WObj:=WO_Pastel;
        MoveL Target_1000,v1000,fine,PortaMarcador\WObj:=WO_Pastel;
        MoveL Target_1010,v1000,fine,PortaMarcador\WObj:=WO_Pastel;
        MoveL Target_1020,v1000,fine,PortaMarcador\WObj:=WO_Pastel;
        MoveL Target_950,v1000,fine,PortaMarcador\WObj:=WO_Pastel;
        MoveL Target_1030,v1000,z100,PortaMarcador\WObj:=WO_Pastel;
    ENDPROC
    PROC Letter_N2()
        MoveL Target_1040,v1000,fine,PortaMarcador\WObj:=WO_Pastel;
        MoveL Target_1050,v1000,fine,PortaMarcador\WObj:=WO_Pastel;
        MoveL Target_1060,v1000,fine,PortaMarcador\WObj:=WO_Pastel;
        MoveL Target_1070,v1000,fine,PortaMarcador\WObj:=WO_Pastel;
        MoveL Target_1080,v1000,fine,PortaMarcador\WObj:=WO_Pastel;
        MoveL Target_1090,v1000,fine,PortaMarcador\WObj:=WO_Pastel;
        MoveL Target_1100,v1000,fine,PortaMarcador\WObj:=WO_Pastel;
        MoveL Target_1110,v1000,fine,PortaMarcador\WObj:=WO_Pastel;
        MoveL Target_1120,v1000,fine,PortaMarcador\WObj:=WO_Pastel;
        MoveL Target_1130,v1000,fine,PortaMarcador\WObj:=WO_Pastel;
        MoveL Target_1040,v1000,fine,PortaMarcador\WObj:=WO_Pastel;
        MoveL Target_1140,v1000,z100,PortaMarcador\WObj:=WO_Pastel;
    ENDPROC
    PROC Letter_I()
        MoveL Target_1150,v1000,fine,PortaMarcador\WObj:=WO_Pastel;
        MoveL Target_1160,v1000,fine,PortaMarcador\WObj:=WO_Pastel;
        MoveL Target_1170,v1000,fine,PortaMarcador\WObj:=WO_Pastel;
        MoveL Target_1180,v1000,fine,PortaMarcador\WObj:=WO_Pastel;
        MoveL Target_1190,v1000,fine,PortaMarcador\WObj:=WO_Pastel;
        MoveL Target_1200,v1000,fine,PortaMarcador\WObj:=WO_Pastel;
        MoveL Target_1210,v1000,fine,PortaMarcador\WObj:=WO_Pastel;
        MoveL Target_1220,v1000,fine,PortaMarcador\WObj:=WO_Pastel;
        MoveL Target_1230,v1000,fine,PortaMarcador\WObj:=WO_Pastel;
        MoveL Target_1240,v1000,fine,PortaMarcador\WObj:=WO_Pastel;
        MoveL Target_1250,v1000,fine,PortaMarcador\WObj:=WO_Pastel;
        MoveL Target_1260,v1000,fine,PortaMarcador\WObj:=WO_Pastel;
        MoveL Target_1150,v1000,fine,PortaMarcador\WObj:=WO_Pastel;
        MoveL Target_1270,v1000,z100,PortaMarcador\WObj:=WO_Pastel;
    ENDPROC
    PROC Home_Sing()
        MoveJ Target_1420,v1000,z100,PortaMarcador\WObj:=wobj0;
        MoveJ Target_1430,v1000,z100,PortaMarcador\WObj:=wobj0;
    ENDPROC
    PROC Sing_Home()
        MoveJ Target_1430,v1000,z100,PortaMarcador\WObj:=wobj0;
        MoveJ Target_1420,v1000,z100,PortaMarcador\WObj:=wobj0;
    ENDPROC
    LOCAL PROC Recorrido()
        MoveJ Target_1420,v150,z100,PortaMarcador\WObj:=wobj0;
        MoveJ Target_1430,v150,z100,PortaMarcador\WObj:=wobj0;
        MoveL Target_10,v100,fine,PortaMarcador\WObj:=WO_Pastel;
        MoveL Target_20,v100,fine,PortaMarcador\WObj:=WO_Pastel;
        MoveL Target_30,v100,fine,PortaMarcador\WObj:=WO_Pastel;
        MoveL Target_40,v100,fine,PortaMarcador\WObj:=WO_Pastel;
        MoveL Target_50,v100,fine,PortaMarcador\WObj:=WO_Pastel;
        MoveL Target_60,v100,fine,PortaMarcador\WObj:=WO_Pastel;
        MoveL Target_70,v100,fine,PortaMarcador\WObj:=WO_Pastel;
        MoveL Target_80,v100,fine,PortaMarcador\WObj:=WO_Pastel;
        MoveL Target_90,v100,fine,PortaMarcador\WObj:=WO_Pastel;
        MoveL Target_100,v100,fine,PortaMarcador\WObj:=WO_Pastel;
        MoveL Target_110,v100,fine,PortaMarcador\WObj:=WO_Pastel;
        MoveL Target_20,v100,fine,PortaMarcador\WObj:=WO_Pastel;
        MoveL Target_1450,v100,z100,PortaMarcador\WObj:=WO_Pastel;
        MoveL Target_1440,v100,z100,PortaMarcador\WObj:=WO_Pastel;
        MoveL Target_130,v100,fine,PortaMarcador\WObj:=WO_Pastel;
        MoveL Target_140,v100,fine,PortaMarcador\WObj:=WO_Pastel;
        MoveC Target_150,Target_160,v100,z100,PortaMarcador\WObj:=WO_Pastel;
        MoveC Target_170,Target_180,v100,z100,PortaMarcador\WObj:=WO_Pastel;
        MoveL Target_190,v100,fine,PortaMarcador\WObj:=WO_Pastel;
        MoveL Target_200,v100,fine,PortaMarcador\WObj:=WO_Pastel;
        MoveC Target_210,Target_220,v100,z100,PortaMarcador\WObj:=WO_Pastel;
        MoveC Target_230,Target_240,v100,z100,PortaMarcador\WObj:=WO_Pastel;
        MoveL Target_250,v100,fine,PortaMarcador\WObj:=WO_Pastel;
        MoveC Target_260,Target_270,v100,z100,PortaMarcador\WObj:=WO_Pastel;
        MoveC Target_280,Target_290,v100,fine,PortaMarcador\WObj:=WO_Pastel;
        MoveL Target_130,v100,fine,PortaMarcador\WObj:=WO_Pastel;
        MoveL Target_300,v100,z100,PortaMarcador\WObj:=WO_Pastel;
        MoveL Target_1480,v100,z100,PortaMarcador\WObj:=WO_Pastel;
        MoveL Target_310,v100,z0,PortaMarcador\WObj:=WO_Pastel;
        MoveL Target_320,v100,fine,PortaMarcador\WObj:=WO_Pastel;
        MoveL Target_330,v100,z100,PortaMarcador\WObj:=WO_Pastel;
        MoveC Target_340,Target_350,v100,z100,PortaMarcador\WObj:=WO_Pastel;
        MoveL Target_360,v100,fine,PortaMarcador\WObj:=WO_Pastel;
        MoveL Target_370,v100,fine,PortaMarcador\WObj:=WO_Pastel;
        MoveL Target_380,v100,z100,PortaMarcador\WObj:=WO_Pastel;
        MoveC Target_390,Target_400,v100,z100,PortaMarcador\WObj:=WO_Pastel;
        MoveL Target_410,v100,fine,PortaMarcador\WObj:=WO_Pastel;
        MoveL Target_420,v100,fine,PortaMarcador\WObj:=WO_Pastel;
        MoveL Target_310,v100,fine,PortaMarcador\WObj:=WO_Pastel;
        MoveL Target_430,v100,z100,PortaMarcador\WObj:=WO_Pastel;
        MoveL Target_1490,v100,z100,PortaMarcador\WObj:=WO_Pastel;
        MoveL Target_440,v100,fine,PortaMarcador\WObj:=WO_Pastel;
        MoveC Target_450,Target_460,v100,z100,PortaMarcador\WObj:=WO_Pastel;
        MoveC Target_470,Target_490,v100,z100,PortaMarcador\WObj:=WO_Pastel;
        MoveL Target_500,v100,z100,PortaMarcador\WObj:=WO_Pastel;
        MoveC Target_510,Target_520,v100,z100,PortaMarcador\WObj:=WO_Pastel;
        MoveC Target_530,Target_550,v100,z100,PortaMarcador\WObj:=WO_Pastel;
        MoveL Target_440,v100,fine,PortaMarcador\WObj:=WO_Pastel;
        MoveL Target_560,v100,z100,PortaMarcador\WObj:=WO_Pastel;
        MoveL Target_1500,v100,z100,PortaMarcador\WObj:=WO_Pastel;
        MoveL Target_570,v100,fine,PortaMarcador\WObj:=WO_Pastel;
        MoveL Target_580,v100,fine,PortaMarcador\WObj:=WO_Pastel;
        MoveL Target_590,v100,fine,PortaMarcador\WObj:=WO_Pastel;
        MoveL Target_600,v100,fine,PortaMarcador\WObj:=WO_Pastel;
        MoveL Target_610,v100,fine,PortaMarcador\WObj:=WO_Pastel;
        MoveL Target_620,v100,fine,PortaMarcador\WObj:=WO_Pastel;
        MoveL Target_630,v100,fine,PortaMarcador\WObj:=WO_Pastel;
        MoveL Target_640,v100,fine,PortaMarcador\WObj:=WO_Pastel;
        MoveL Target_650,v100,fine,PortaMarcador\WObj:=WO_Pastel;
        MoveL Target_660,v100,fine,PortaMarcador\WObj:=WO_Pastel;
        MoveL Target_570,v100,fine,PortaMarcador\WObj:=WO_Pastel;
        MoveL Target_670,v100,z100,PortaMarcador\WObj:=WO_Pastel;
        MoveL Target_1510,v100,z100,PortaMarcador\WObj:=WO_Pastel;
        MoveL Target_680,v100,fine,PortaMarcador\WObj:=WO_Pastel;
        MoveL Target_690,v100,fine,PortaMarcador\WObj:=WO_Pastel;
        MoveL Target_700,v100,fine,PortaMarcador\WObj:=WO_Pastel;
        MoveL Target_710,v100,fine,PortaMarcador\WObj:=WO_Pastel;
        MoveL Target_720,v100,fine,PortaMarcador\WObj:=WO_Pastel;
        MoveL Target_730,v100,fine,PortaMarcador\WObj:=WO_Pastel;
        MoveL Target_740,v100,fine,PortaMarcador\WObj:=WO_Pastel;
        MoveL Target_750,v100,fine,PortaMarcador\WObj:=WO_Pastel;
        MoveL Target_680,v100,fine,PortaMarcador\WObj:=WO_Pastel;
        MoveL Target_760,v100,fine,PortaMarcador\WObj:=WO_Pastel;
        MoveL Target_1520,v100,z100,PortaMarcador\WObj:=WO_Pastel;
        MoveL Target_770,v100,fine,PortaMarcador\WObj:=WO_Pastel;
        MoveL Target_780,v100,fine,PortaMarcador\WObj:=WO_Pastel;
        MoveL Target_790,v100,fine,PortaMarcador\WObj:=WO_Pastel;
        MoveL Target_800,v100,fine,PortaMarcador\WObj:=WO_Pastel;
        MoveL Target_810,v100,fine,PortaMarcador\WObj:=WO_Pastel;
        MoveL Target_820,v100,fine,PortaMarcador\WObj:=WO_Pastel;
        MoveL Target_830,v100,fine,PortaMarcador\WObj:=WO_Pastel;
        MoveL Target_840,v100,fine,PortaMarcador\WObj:=WO_Pastel;
        MoveL Target_770,v100,fine,PortaMarcador\WObj:=WO_Pastel;
        MoveL Target_850,v100,z100,PortaMarcador\WObj:=WO_Pastel;
        MoveL Target_1530,v100,z100,PortaMarcador\WObj:=WO_Pastel;
        MoveL Target_860,v100,fine,PortaMarcador\WObj:=WO_Pastel;
        MoveL Target_870,v100,fine,PortaMarcador\WObj:=WO_Pastel;
        MoveC Target_880,Target_890,v100,fine,PortaMarcador\WObj:=WO_Pastel;
        MoveL Target_900,v100,fine,PortaMarcador\WObj:=WO_Pastel;
        MoveC Target_910,Target_920,v100,fine,PortaMarcador\WObj:=WO_Pastel;
        MoveL Target_930,v100,fine,PortaMarcador\WObj:=WO_Pastel;
        MoveL Target_860,v100,fine,PortaMarcador\WObj:=WO_Pastel;
        MoveL Target_940,v100,z100,PortaMarcador\WObj:=WO_Pastel;
        MoveL Target_1540,v100,z100,PortaMarcador\WObj:=WO_Pastel;
        MoveL Target_950,v100,fine,PortaMarcador\WObj:=WO_Pastel;
        MoveL Target_960,v100,fine,PortaMarcador\WObj:=WO_Pastel;
        MoveL Target_970,v100,fine,PortaMarcador\WObj:=WO_Pastel;
        MoveL Target_980,v100,fine,PortaMarcador\WObj:=WO_Pastel;
        MoveL Target_990,v100,fine,PortaMarcador\WObj:=WO_Pastel;
        MoveL Target_1000,v100,fine,PortaMarcador\WObj:=WO_Pastel;
        MoveL Target_1550,v100,z100,PortaMarcador\WObj:=WO_Pastel;
        MoveL Target_1010,v100,fine,PortaMarcador\WObj:=WO_Pastel;
        MoveL Target_1020,v100,fine,PortaMarcador\WObj:=WO_Pastel;
        MoveL Target_950,v100,fine,PortaMarcador\WObj:=WO_Pastel;
        MoveL Target_1030,v100,z100,PortaMarcador\WObj:=WO_Pastel;
        MoveL Target_1550,v100,z100,PortaMarcador\WObj:=WO_Pastel;
        MoveL Target_1040,v100,fine,PortaMarcador\WObj:=WO_Pastel;
        MoveL Target_1050,v100,fine,PortaMarcador\WObj:=WO_Pastel;
        MoveL Target_1060,v100,fine,PortaMarcador\WObj:=WO_Pastel;
        MoveL Target_1070,v100,fine,PortaMarcador\WObj:=WO_Pastel;
        MoveL Target_1080,v100,fine,PortaMarcador\WObj:=WO_Pastel;
        MoveL Target_1090,v100,fine,PortaMarcador\WObj:=WO_Pastel;
        MoveL Target_1110,v100,fine,PortaMarcador\WObj:=WO_Pastel;
        MoveL Target_1120,v100,fine,PortaMarcador\WObj:=WO_Pastel;
        MoveL Target_1100,v100,fine,PortaMarcador\WObj:=WO_Pastel;
        MoveL Target_1130,v100,fine,PortaMarcador\WObj:=WO_Pastel;
        MoveL Target_1040,v100,fine,PortaMarcador\WObj:=WO_Pastel;
        MoveL Target_1140,v100,z100,PortaMarcador\WObj:=WO_Pastel;
        MoveL Target_1270,v100,z100,PortaMarcador\WObj:=WO_Pastel;
        MoveL Target_1150_2,v100,fine,PortaMarcador\WObj:=WO_Pastel;
        MoveL Target_1160_2,v100,fine,PortaMarcador\WObj:=WO_Pastel;
        MoveL Target_1170_2,v100,fine,PortaMarcador\WObj:=WO_Pastel;
        MoveL Target_1180_2,v100,fine,PortaMarcador\WObj:=WO_Pastel;
        MoveL Target_1190_2,v100,fine,PortaMarcador\WObj:=WO_Pastel;
        MoveL Target_1200_2,v100,fine,PortaMarcador\WObj:=WO_Pastel;
        MoveL Target_1210_2,v100,fine,PortaMarcador\WObj:=WO_Pastel;
        MoveL Target_1220_2,v100,fine,PortaMarcador\WObj:=WO_Pastel;
        MoveL Target_1230_2,v100,fine,PortaMarcador\WObj:=WO_Pastel;
        MoveL Target_1240_2,v100,fine,PortaMarcador\WObj:=WO_Pastel;
        MoveL Target_1250_2,v100,fine,PortaMarcador\WObj:=WO_Pastel;
        MoveL Target_1260_2,v100,fine,PortaMarcador\WObj:=WO_Pastel;
        MoveL Target_1150_2,v100,fine,PortaMarcador\WObj:=WO_Pastel;
        MoveL Target_1270_2,v100,z100,PortaMarcador\WObj:=WO_Pastel;
        MoveL Target_1560,v100,z100,PortaMarcador\WObj:=WO_Pastel;
        MoveL Target_1280_2,v100,z100,PortaMarcador\WObj:=WO_Pastel;
        MoveL Target_1290_2,v100,fine,PortaMarcador\WObj:=WO_Pastel;
        MoveL Target_1300_2,v100,fine,PortaMarcador\WObj:=WO_Pastel;
        MoveL Target_1310_2,v100,fine,PortaMarcador\WObj:=WO_Pastel;
        MoveL Target_1320_2,v100,fine,PortaMarcador\WObj:=WO_Pastel;
        MoveL Target_1330_2,v100,fine,PortaMarcador\WObj:=WO_Pastel;
        MoveL Target_1340_2,v100,fine,PortaMarcador\WObj:=WO_Pastel;
        MoveL Target_1350_2,v100,fine,PortaMarcador\WObj:=WO_Pastel;
        MoveL Target_1360_2,v100,fine,PortaMarcador\WObj:=WO_Pastel;
        MoveL Target_1370_2,v100,fine,PortaMarcador\WObj:=WO_Pastel;
        MoveL Target_1380_2,v100,fine,PortaMarcador\WObj:=WO_Pastel;
        MoveL Target_1390_2,v100,z100,PortaMarcador\WObj:=WO_Pastel;
        MoveL Target_1280_2,v100,z100,PortaMarcador\WObj:=WO_Pastel;
        MoveJ Target_1430,v1000,z100,PortaMarcador\WObj:=wobj0;
        MoveJ Target_1420,v1000,z100,PortaMarcador\WObj:=wobj0;
    ENDPROC
    LOCAL PROC Maintenance()
        MoveJ Target_1420,v1000,z100,PortaMarcador\WObj:=wobj0;
        MoveJ Mantenimiento,v1000,z100,PortaMarcador\WObj:=wobj0;
    ENDPROC
ENDMODULE
